FUNCTION_BLOCK FB_Waermezaehler_WP
VAR_INPUT
	Telegramm	: ARRAY[1..cMBUS_MaxTelegrams] OF ST_MBus_Data2;

END_VAR
VAR_IN_OUT
	Zustand		: ST_WZ_Zustand;
END_VAR
VAR
END_VAR
VAR // added by the converter: edge detectors and wires of the graphical bodies
    _w1, _w2, _w3 : ANY;
END_VAR

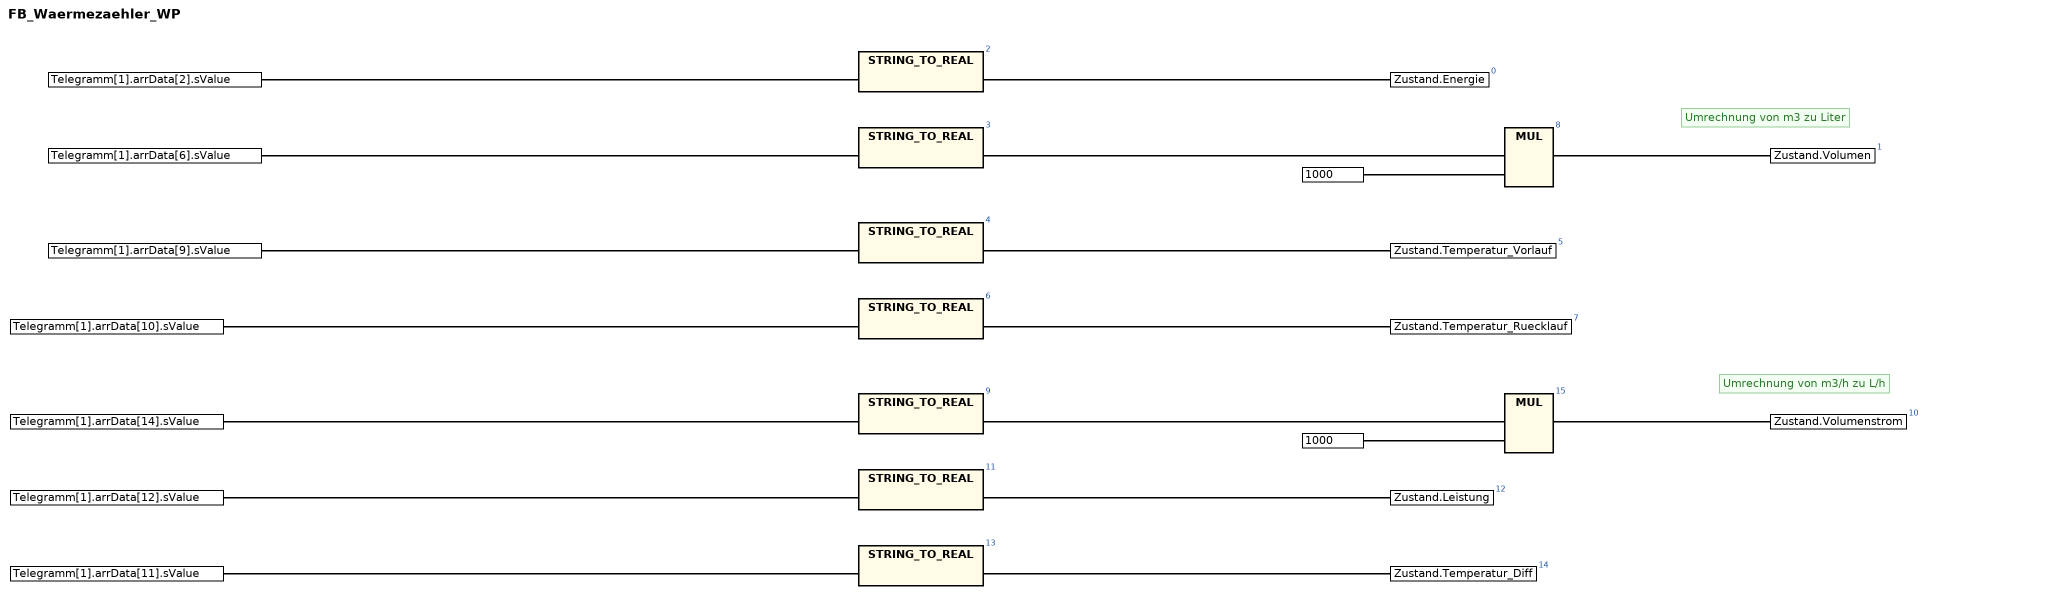
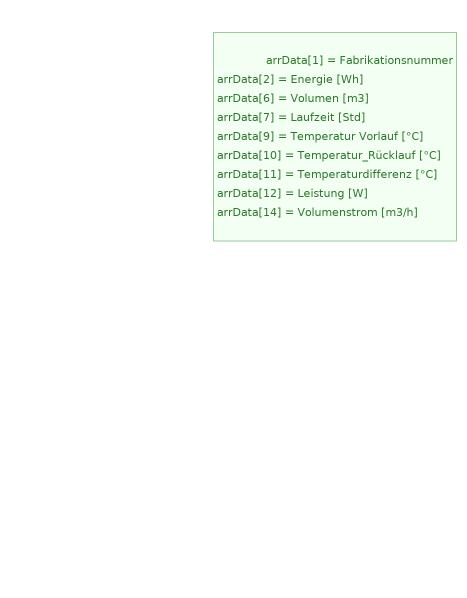
Zustand.Energie := _w1;
// 							arrData[1] = Fabrikationsnummer
// arrData[2] = Energie [Wh]
// arrData[6] = Volumen [m3]
// arrData[7] = Laufzeit [Std]
// arrData[9] = Temperatur Vorlauf [°C]
// arrData[10] = Temperatur_Rücklauf [°C]
// arrData[11] = Temperaturdifferenz [°C]
// arrData[12] = Leistung [W]
// arrData[14] = Volumenstrom [m3/h]
//
// Umrechnung von m3 zu Liter
Zustand.Volumen := _w2;
_w1 := STRING_TO_REAL(Telegramm[1].arrData[2].sValue);
Zustand.Temperatur_Vorlauf := STRING_TO_REAL(Telegramm[1].arrData[9].sValue);
Zustand.Temperatur_Ruecklauf := STRING_TO_REAL(Telegramm[1].arrData[10].sValue);
_w2 := STRING_TO_REAL(Telegramm[1].arrData[6].sValue) * 1000;
// Umrechnung von m3/h zu L/h
Zustand.Volumenstrom := _w3;
Zustand.Leistung := STRING_TO_REAL(Telegramm[1].arrData[12].sValue);
Zustand.Temperatur_Diff := STRING_TO_REAL(Telegramm[1].arrData[11].sValue);
_w3 := STRING_TO_REAL(Telegramm[1].arrData[14].sValue) * 1000;

END_FUNCTION_BLOCK

(* stored: Version 1.1.0.1, ProductVersion 3.1.4024.9
   POU FB_Waermezaehler_WP: Id {2d46c6a0-ac39-4ee3-b544-dcc391aaeade}, SpecialFunc None *)
